INTERFACE I_PackMLStateActionProvider

METHOD PROTECTED H_OnAborted
VAR_INPUT
	bFirstScan	: BOOL;
END_VAR
END_METHOD

METHOD PROTECTED H_OnAborting : E_PackMLHookResult
VAR_INPUT
	bFirstScan	: BOOL;
END_VAR
END_METHOD

METHOD PROTECTED H_OnClearing : E_PackMLHookResult
VAR_INPUT
	bFirstScan	: BOOL;
END_VAR
END_METHOD

METHOD PROTECTED H_OnComplete
VAR_INPUT
	bFirstScan	: BOOL;
END_VAR
END_METHOD

METHOD PROTECTED H_OnCompleting : E_PackMLHookResult
VAR_INPUT
	bFirstScan	: BOOL;
END_VAR
END_METHOD

METHOD PROTECTED H_OnExecute : E_PackMLHookResult
VAR_INPUT
	bFirstScan	: BOOL;
END_VAR
END_METHOD

METHOD PROTECTED H_OnHeld
VAR_INPUT
	bFirstScan	: BOOL;
END_VAR
END_METHOD

METHOD PROTECTED H_OnHolding : E_PackMLHookResult
VAR_INPUT
	bFirstScan	: BOOL;
END_VAR
END_METHOD

METHOD PROTECTED H_OnIdle
VAR_INPUT
	bFirstScan	: BOOL;
END_VAR
END_METHOD

METHOD PROTECTED H_OnResetting : E_PackMLHookResult
VAR_INPUT
	bFirstScan	: BOOL;
END_VAR
END_METHOD

METHOD PROTECTED H_OnStarting : E_PackMLHookResult
VAR_INPUT
	bFirstScan	: BOOL;
END_VAR
END_METHOD

METHOD PROTECTED H_OnStopped
VAR_INPUT
	bFirstScan	: BOOL;
END_VAR
END_METHOD

METHOD PROTECTED H_OnStopping : E_PackMLHookResult
VAR_INPUT
	bFirstScan	: BOOL;
END_VAR
END_METHOD

METHOD PROTECTED H_OnSuspended
VAR_INPUT
	bFirstScan	: BOOL;
END_VAR
END_METHOD

METHOD PROTECTED H_OnSuspending : E_PackMLHookResult
VAR_INPUT
	bFirstScan	: BOOL;
END_VAR
END_METHOD

METHOD PROTECTED H_OnUndefined : E_PackMLHookResult
VAR_INPUT
	bFirstScan	: BOOL;
END_VAR
END_METHOD

METHOD PROTECTED H_OnUnholding : E_PackMLHookResult
VAR_INPUT
	bFirstScan	: BOOL;
END_VAR
END_METHOD

METHOD PROTECTED H_OnUnsuspending : E_PackMLHookResult
VAR_INPUT
	bFirstScan	: BOOL;
END_VAR
END_METHOD

END_INTERFACE

(* stored: Version 1.1.0.1, ProductVersion 3.1.4026.18
   Itf I_PackMLStateActionProvider: Id {b0c61b72-0d64-4968-b250-19f75305f691}
   Method H_OnAborted: Id {8236ef7b-4242-46c2-8c5b-bc5f877ae3ad}
   Method H_OnAborting: Id {0293a339-2d80-49c1-b8b7-c2ade899c2b5}
   Method H_OnClearing: Id {2a5a74a1-eca6-47fc-aa70-4518b319616d}
   Method H_OnComplete: Id {cb05bd86-e8e7-48a7-8b99-2d8626e3b671}
   Method H_OnCompleting: Id {28f6613a-d74e-4079-96e8-b6d3cc93f8f8}
   Method H_OnExecute: Id {4fde2c9f-1bc0-40d8-8000-d1389dbfe797}
   Method H_OnHeld: Id {8bd117dd-eec3-4641-a050-d0eebc67b42a}
   Method H_OnHolding: Id {ae3e8ccd-c5eb-4c62-b17c-2c92691d80db}
   Method H_OnIdle: Id {542ef73c-af0b-412c-8f9f-63dcb19fc589}
   Method H_OnResetting: Id {4262849a-1400-4113-ad7a-47b2800c7d4c}
   Method H_OnStarting: Id {b69a6263-9905-4e0b-a8af-fb10f7b1db4a}
   Method H_OnStopped: Id {0fe7eee7-b063-49fb-97c2-6df17165d16f}
   Method H_OnStopping: Id {34c5ef02-9d8f-4722-86e9-c4f7a9d6ca33}
   Method H_OnSuspended: Id {f8a71111-3b51-4224-8d42-1c1291102b73}
   Method H_OnSuspending: Id {99b5d2bf-e0dd-4e8c-a9fc-a067f5e7fc1b}
   Method H_OnUndefined: Id {bbe8bbd5-0e39-4a21-a946-c90a6bc2475a}
   Method H_OnUnholding: Id {9bab317c-68d8-4938-8976-39c927e25752}
   Method H_OnUnsuspending: Id {6bffe64a-fd6d-4b25-9400-fe92a4fb9a62} *)
